ABB RobotStudio station: proiect_1301A_Nichifor_Cristian_Musteata_Valeriu.rspag

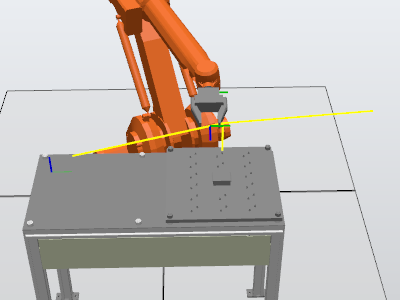
--- station ---
Station pikplace (saved by RobotStudio 25.4.11475.0)
Controller R1400, task T_ROB1: task frame (RAPID world) sits at (0, 0, 0) mm, rotated rx 0 ry 0 rz -45 deg in the station
Controller R1400
  mechanical unit ROB_1: IRB1400_5_144__01, 6 joints, base frame (0, 0, 0) mm
Layout (positions relative to the parent item):
  - IRB1400_5_144__01 [mechanism, from Robots\IRB1400_5_144__01.rslib] at (0, 0, 0) mm, rotated rx 0 ry 0 rz -45 deg; joint values [-0.3822, -0.6501, 0.0834, -1.4092, 0.4046, 1.4548] (rad or m)
  - Gripper_R1400 [smart component, from Components\Gripper_R1400.rslib] at (201.82, -557.27, 1000.36) mm, rotated rx 180 ry 81.97 rz 90 deg
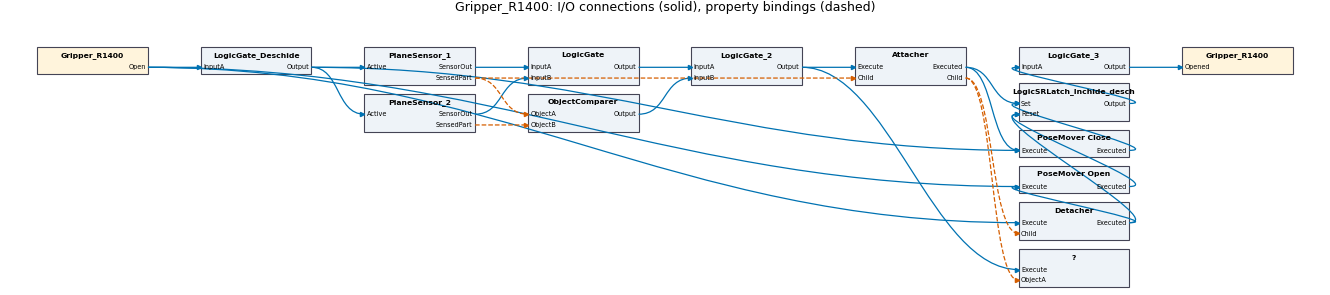
      connections:
        Attacher.Executed -> LogicSRLatch_Inchide_deschide.Set
        Detacher.Executed -> LogicSRLatch_Inchide_deschide.Reset
        Attacher.Executed -> PoseMover Close.Execute
        PoseMover Close.Executed -> LogicSRLatch_Inchide_deschide.Set
        Detacher.Executed -> PoseMover Open.Execute
        PoseMover Open.Executed -> LogicSRLatch_Inchide_deschide.Reset
        LogicGate.Output -> LogicGate_2.InputA
        ObjectComparer.Output -> LogicGate_2.InputB
        LogicGate_2.Output -> ?.Execute
        LogicGate_2.Output -> Attacher.Execute
        PlaneSensor_1.SensorOut -> LogicGate.InputA
        PlaneSensor_2.SensorOut -> LogicGate.InputB
        LogicGate_Deschide.Output -> PlaneSensor_2.Active
        LogicGate_Deschide.Output -> PlaneSensor_1.Active
        LogicGate_Deschide.Output -> PoseMover Close.Execute
        LogicSRLatch_Inchide_deschide.Output -> LogicGate_3.InputA
        LogicGate_3.Output -> Gripper_R1400.Opened
        Gripper_R1400.Open -> LogicGate_Deschide.InputA
        Gripper_R1400.Open -> Detacher.Execute
        Gripper_R1400.Open -> PoseMover Open.Execute
        Attacher.Child => Detacher.Child
        Attacher.Child => ?.ObjectA
        PlaneSensor_1.SensedPart => Attacher.Child
        PlaneSensor_1.SensedPart => ObjectComparer.ObjectA
        PlaneSensor_2.SensedPart => ObjectComparer.ObjectB
    - Attacher [smart component, from Components\Gripper_R1400.rslib]
        properties: Parent=Gripper; Flange=0; Child=(none); Mount=false; Offset=[0 0 0]; Orientation=[0 0 0]
    - Detacher [smart component, from Components\Gripper_R1400.rslib]
        properties: Child=(none); KeepPosition=true
    - LogicGate_Deschide [smart component, from Components\Gripper_R1400.rslib]
        properties: Operator=NOT; Delay=0
    - LogicSRLatch_Inchide_deschide [smart component, from Components\Gripper_R1400.rslib]
    - PoseMover Close [smart component, from Components\Gripper_R1400.rslib]
        properties: Mechanism=Gripper; Pose=3; Duration=0
    - PoseMover Open [smart component, from Components\Gripper_R1400.rslib]
        properties: Mechanism=Gripper; Pose=2; Duration=0
    - ObjectComparer [smart component, from Components\ObjectComparer.rslib]
        properties: ObjectA=(none); ObjectB=(none)
    - LogicGate [smart component, from Components\LogicGate.rslib]
        properties: Operator=AND; Delay=0
    - LogicGate_2 [smart component, from Components\LogicGate.rslib]
        properties: Operator=AND; Delay=0
    - PlaneSensor_1 [smart component, from Components\PlaneSensor.rslib]
        properties: Origin=[-0.015 0.03 0.128]; Axis1=[0 0 0.055]; Axis2=[0.03 0 0]; SensedPart=(none); SenseMultiple=false; Tag=(none)
      - _sensorPart_ [part], size 30 x 0 x 55 mm
    - PlaneSensor_2 [smart component, from Components\PlaneSensor.rslib]
        properties: Origin=[-0.015 -0.03 0.128]; Axis1=[0 0 0.055]; Axis2=[0.03 0 0]; SensedPart=(none); SenseMultiple=false; Tag=(none)
      - _sensorPart_ [part], size 30 x 0 x 55 mm
    - Gripper [mechanism, from Components\Gripper_R1400.rslib] at (0, 0.03, 0) mm; joint values [0.0105, -0.0105] (rad or m)
    - LogicGate_3 [smart component, from Components\LogicGate.rslib]
        properties: Operator=NOT; Delay=0
  - Paleta [part, from Components\Paleta.rslib] at (240, -878, 808) mm, rotated rx 0 ry 0 rz -90 deg
  - Stoc1400 [smart component, from Components\Stoc1400.rslib] at (0, -878, 0) mm, rotated rx 0 ry 0 rz -90 deg
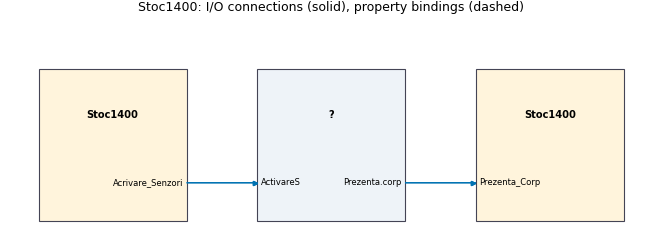
      connections:
        Stoc1400.Acrivare_Senzori -> ?.ActivareS
        Stoc1400.Acrivare_Senzori -> ?.ActivareS
        ?.Prezenta.corp -> Stoc1400.Prezenta_Corp
        ?.Prezenta.corp -> Stoc1400.Prezenta_Corp
    - 679#Body 1 [part, from Components\Stoc1400.rslib]
    - 681#Body 2 [part, from Components\Stoc1400.rslib]
    - 683#Body 3 [part, from Components\Stoc1400.rslib]
    - 685#Body 4 [part, from Components\Stoc1400.rslib]
    - 687#Body 5 [part, from Components\Stoc1400.rslib]
    - 689#Body 6 [part, from Components\Stoc1400.rslib]
    - 691#Body 7 [part, from Components\Stoc1400.rslib]
    - 693#Body 8 [part, from Components\Stoc1400.rslib]
    - 695#Body 9 [part, from Components\Stoc1400.rslib]
    - 697#Body 10 [part, from Components\Stoc1400.rslib]
    - 701#Body 12 [part, from Components\Stoc1400.rslib]
    - 703#Body 13 [part, from Components\Stoc1400.rslib]
    - 705#Body 14 [part, from Components\Stoc1400.rslib]
    - 707#Body 15 [part, from Components\Stoc1400.rslib]
    - 755#Body 39 [part, from Components\Stoc1400.rslib]
    - 757#Body 40 [part, from Components\Stoc1400.rslib]
    - 759#Body 41 [part, from Components\Stoc1400.rslib]
    - 761#Body 42 [part, from Components\Stoc1400.rslib]
    - 785#Body 54 [part, from Components\Stoc1400.rslib]
    - 787#Body 55 [part, from Components\Stoc1400.rslib]
    - 789#Body 56 [part, from Components\Stoc1400.rslib]
    - 791#Body 57 [part, from Components\Stoc1400.rslib]
    - 793#Body 58 [part, from Components\Stoc1400.rslib]
    - Part [part, from Components\Stoc1400.rslib]
    - Part_2 [part, from Components\Stoc1400.rslib]
    - Part_3 [part, from Components\Stoc1400.rslib]
    - Part_4 [part, from Components\Stoc1400.rslib]
Attachment: Gripper_R1400 is attached to IRB1400_5_144__01 / Link6
Station logic (signal -> signal, property => property):
  R1400.DO10_9 -> Gripper_R1400.Open
Targets, tools, work objects and paths stored in the station and not in the controller backup, written as RAPID:
! task T_ROB1
MODULE Module1
  PROC ZERO()
    MoveL T0_1,v200,fine,Efector\WObj:=Workobject_1;
    MoveC T0_2,T0_3,v200,fine,Efector\WObj:=Workobject_1;
    MoveC T0_4,T0_1,v200,fine,Efector\WObj:=Workobject_1;
    MoveL ref,v200,fine,Efector\WObj:=Workobject_1;
  ENDPROC
  PROC ONE()
    MoveL T1_1,v200,fine,Efector\WObj:=Workobject_1;
    MoveL T1_2,v200,fine,Efector\WObj:=Workobject_1;
    MoveL T1_3,v200,fine,Efector\WObj:=Workobject_1;
    MoveL ref,v200,fine,Efector\WObj:=Workobject_1;
  ENDPROC
  PROC TWO()
    MoveL T2_1,v200,fine,Efector\WObj:=Workobject_1;
    MoveC T2_2,T2_3,v200,fine,Efector\WObj:=Workobject_1;
    MoveL T2_4,v200,fine,Efector\WObj:=Workobject_1;
    MoveL T2_5,v200,fine,Efector\WObj:=Workobject_1;
    MoveL ref,v200,fine,Efector\WObj:=Workobject_1;
  ENDPROC
  PROC THREE()
    MoveL T3_1,v200,fine,Efector\WObj:=Workobject_1;
    MoveL T3_2,v200,fine,Efector\WObj:=Workobject_1;
    MoveL T3_3,v200,fine,Efector\WObj:=Workobject_1;
    MoveC T3_4,T3_5,v200,fine,Efector\WObj:=Workobject_1;
    MoveL ref,v200,fine,Efector\WObj:=Workobject_1;
  ENDPROC
  PROC FOUR()
    MoveL T4_1,v200,fine,Efector\WObj:=Workobject_1;
    MoveL T4_2,v200,fine,Efector\WObj:=Workobject_1;
    MoveL T4_3,v200,fine,Efector\WObj:=Workobject_1;
    MoveL T4_4,v200,fine,Efector\WObj:=Workobject_1;
    MoveL ref,v200,fine,Efector\WObj:=Workobject_1;
  ENDPROC
  PROC NINE()
    MoveL T9_1,v200,fine,Efector\WObj:=Workobject_1;
    MoveC T9_2,T9_3,v200,fine,Efector\WObj:=Workobject_1;
    MoveL T9_4,v200,fine,Efector\WObj:=Workobject_1;
    MoveC T9_5,T9_6,v200,fine,Efector\WObj:=Workobject_1;
    MoveC T9_7,T9_4,v200,fine,Efector\WObj:=Workobject_1;
    MoveL ref,v200,fine,Efector\WObj:=Workobject_1;
  ENDPROC
  PROC SIX()
    MoveL T6_1,v200,fine,Efector\WObj:=Workobject_1;
    MoveC T6_2,T6_3,v200,fine,Efector\WObj:=Workobject_1;
    MoveL T6_4,v200,fine,Efector\WObj:=Workobject_1;
    MoveC T6_5,T6_6,v200,fine,Efector\WObj:=Workobject_1;
    MoveC T6_7,T6_4,v200,fine,Efector\WObj:=Workobject_1;
    MoveL ref,v200,fine,Efector\WObj:=Workobject_1;
  ENDPROC
  PROC FIVE()
    MoveL T5_1,v200,fine,Efector\WObj:=Workobject_1;
    MoveL T5_2,v200,fine,Efector\WObj:=Workobject_1;
    MoveL T5_3,v200,fine,Efector\WObj:=Workobject_1;
    MoveC T5_4,T5_5,v200,fine,Efector\WObj:=Workobject_1;
    MoveL ref,v200,fine,Efector\WObj:=Workobject_1;
  ENDPROC
  PROC SEVEN()
    MoveL T7_1,v200,fine,Efector\WObj:=Workobject_1;
    MoveL T7_2,v200,fine,Efector\WObj:=Workobject_1;
    MoveL T7_3,v200,fine,Efector\WObj:=Workobject_1;
    MoveL ref,v200,fine,Efector\WObj:=Workobject_1;
  ENDPROC
  PROC EIGHT()
    MoveL T8_1,v200,fine,Efector\WObj:=Workobject_1;
    MoveC T8_2,T8_3,v200,fine,Efector\WObj:=Workobject_1;
    MoveC T8_4,T8_5,v200,fine,Efector\WObj:=Workobject_1;
    MoveC T8_6,T8_3,v200,fine,Efector\WObj:=Workobject_1;
    MoveC T8_7,T8_1,v200,fine,Efector\WObj:=Workobject_1;
    MoveL ref,v200,fine,Efector\WObj:=Workobject_1;
  ENDPROC
ENDMODULE


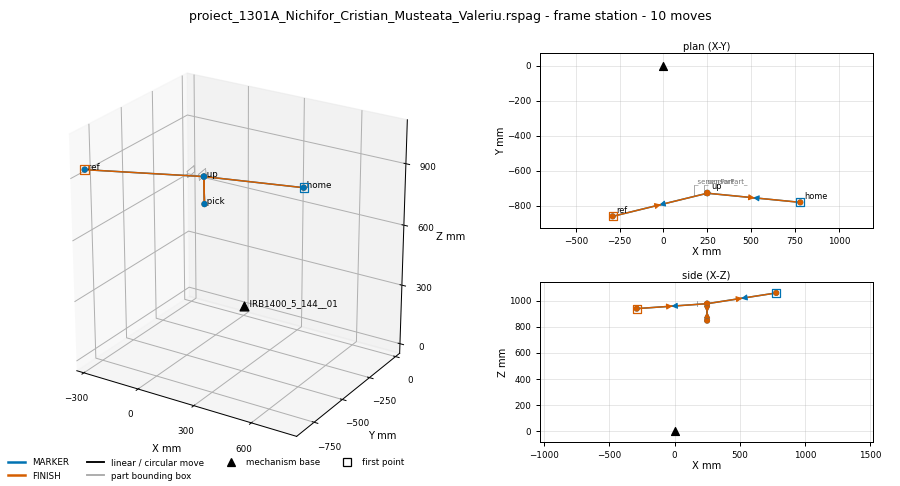
[picture p0: tool path of proiect_1301A_Nichifor_Cristian_Musteata_Valeriu.rspag in frame station, 10 of 60 moves have a stored position in this frame; points joined in program order, loops and branches not executed]
--- Controller Data/R1400/RAPID/TASK1/PROGMOD/Module1.mod ---
MODULE Module1
    PERS tooldata Efector:=[TRUE,[[0,0.033033672,184.3],[1,0,0,0]],[1.5,[0,0,90],[1,0,0,0],0.01,0.01,0.01]];
    PERS wobjdata Workobject_1:=[FALSE,TRUE,"",[[276.123735704,-827.667234537,798.663444233],[0.923877305,0.000104396,-0.002651392,-0.382679612]],[[0,0,0],[1,0,0,0]]];
    CONST robtarget home:=[[0.834488103,1170.696929347,259.084700159],[0.459642479,-0.331462463,0.801426912,0.191249396],[-1,0,-1,0],[9E+09,9E+09,9E+09,9E+09,9E+09,9E+09]];
    CONST robtarget up:=[[-51.633208179,640.397645531,178.164826806],[0.705400436,-0.000783768,0.708808148,-0.000787554],[-1,-2,1,0],[9E+09,9E+09,9E+09,9E+09,9E+09,9E+09]];
    CONST robtarget pick:=[[-55.259706896,640.108764023,48.166657408],[0.705400436,-0.000783768,0.708808148,-0.000787554],[-1,-2,1,0],[9E+09,9E+09,9E+09,9E+09,9E+09,9E+09]];
    CONST robtarget ref:=[[80.028130577,100.720123453,140.72904745],[0.002409616,-0.000002677,-0.99999648,0.001111092],[-1,0,-1,0],[9E+09,9E+09,9E+09,9E+09,9E+09,9E+09]];
CONST robtarget T0_1:=[[9.546208479,100.497907125,40.730455604],[0.002409616,-0.000002677,-0.99999648,0.001111092],[-1,-1,0,0],[9E+09,9E+09,9E+09,9E+09,9E+09,9E+09]];
    CONST robtarget T0_2:=[[41.035842809,79.777621062,40.624742502],[0.002409616,-0.000002677,-0.99999648,0.001111092],[-1,-1,0,0],[9E+09,9E+09,9E+09,9E+09,9E+09,9E+09]];
    CONST robtarget T0_3:=[[81.732370203,107.749116179,40.366456021],[0.002409616,-0.000002677,-0.99999648,0.001111092],[-1,-1,0,0],[9E+09,9E+09,9E+09,9E+09,9E+09,9E+09]];
    CONST robtarget T0_4:=[[36.187899089,125.180560875,40.547211878],[0.002409616,-0.000002677,-0.99999648,0.001111092],[-1,-1,0,0],[9E+09,9E+09,9E+09,9E+09,9E+09,9E+09]];
    CONST robtarget T1_1:=[[23.778043214,86.267789909,40.693490346],[0.002409616,-0.000002677,-0.99999648,0.001111093],[-1,0,-1,0],[9E+09,9E+09,9E+09,9E+09,9E+09,9E+09]];
    CONST robtarget T1_2:=[[8.731217939,99.845917516,40.735832074],[0.002409616,-0.000002677,-0.99999648,0.001111093],[-1,0,-1,0],[9E+09,9E+09,9E+09,9E+09,9E+09,9E+09]];
    CONST robtarget T1_3:=[[80.636382929,100.842145042,40.387086501],[0.002409616,-0.000002677,-0.99999648,0.001111093],[-1,0,-1,0],[9E+09,9E+09,9E+09,9E+09,9E+09,9E+09]];
    CONST robtarget T2_1:=[[31.755950553,80.841717855,40.667100297],[0.002409616,-0.000002677,-0.99999648,0.001111093],[-1,0,-1,0],[9E+09,9E+09,9E+09,9E+09,9E+09,9E+09]];
    CONST robtarget T2_2:=[[6.08624864,99.311947147,40.74976553],[0.002409616,-0.000002677,-0.99999648,0.001111093],[-1,0,-1,0],[9E+09,9E+09,9E+09,9E+09,9E+09,9E+09]];
    CONST robtarget T2_3:=[[29.104981321,125.470636052,40.580701845],[0.002409616,-0.000002677,-0.99999648,0.001111093],[-1,0,-1,0],[9E+09,9E+09,9E+09,9E+09,9E+09,9E+09]];
    CONST robtarget T2_4:=[[71.480489244,86.448278602,40.463197375],[0.002409616,-0.000002677,-0.99999648,0.001111093],[-1,0,-1,0],[9E+09,9E+09,9E+09,9E+09,9E+09,9E+09]];
    CONST robtarget T2_5:=[[70.80349709,127.872183573,40.374407927],[0.002409616,-0.000002677,-0.99999648,0.001111093],[-1,0,-1,0],[9E+09,9E+09,9E+09,9E+09,9E+09,9E+09]];
    CONST robtarget T3_1:=[[18.710215411,82.591773594,40.726082499],[0.002409616,-0.000002677,-0.99999648,0.001111093],[-1,0,-1,0],[9E+09,9E+09,9E+09,9E+09,9E+09,9E+09]];
    CONST robtarget T3_2:=[[19.688090682,111.187772163,40.657823899],[0.002409616,-0.000002677,-0.99999648,0.001111093],[-1,0,-1,0],[9E+09,9E+09,9E+09,9E+09,9E+09,9E+09]];
    CONST robtarget T3_3:=[[45.419791871,103.366515913,40.55119576],[0.002409616,-0.000002677,-0.99999648,0.001111093],[-1,0,-1,0],[9E+09,9E+09,9E+09,9E+09,9E+09,9E+09]];
    CONST robtarget T3_4:=[[68.022529389,116.554241299,40.41296091],[0.002409616,-0.000002677,-0.99999648,0.001111093],[-1,0,-1,0],[9E+09,9E+09,9E+09,9E+09,9E+09,9E+09]];
    CONST robtarget T3_5:=[[73.635464218,90.505245507,40.443796548],[0.002409616,-0.000002677,-0.99999648,0.001111093],[-1,0,-1,0],[9E+09,9E+09,9E+09,9E+09,9E+09,9E+09]];
    CONST robtarget T4_1:=[[53.83069419,124.165374487,40.464442032],[0.002409616,-0.000002677,-0.99999648,0.001111093],[-1,0,-1,0],[9E+09,9E+09,9E+09,9E+09,9E+09,9E+09]];
    CONST robtarget T4_2:=[[53.075702975,80.033491537,40.566150282],[0.002409616,-0.000002677,-0.99999648,0.001111093],[-1,0,-1,0],[9E+09,9E+09,9E+09,9E+09,9E+09,9E+09]];
    CONST robtarget T4_3:=[[9.18787321,109.525888713,40.712120516],[0.002409616,-0.000002677,-0.99999648,0.001111093],[-1,0,-1,0],[9E+09,9E+09,9E+09,9E+09,9E+09,9E+09]];
    CONST robtarget T4_4:=[[83.035355052,110.99609425,40.352961057],[0.002409616,-0.000002677,-0.99999648,0.001111093],[-1,0,-1,0],[9E+09,9E+09,9E+09,9E+09,9E+09,9E+09]];
    CONST robtarget T9_1:=[[70.611499337,82.764297004,40.475571821],[0.002409616,-0.000002677,-0.99999648,0.001111093],[-1,0,-1,0],[9E+09,9E+09,9E+09,9E+09,9E+09,9E+09]];
    CONST robtarget T9_2:=[[86.448315421,103.968075054,40.352130656],[0.002409616,-0.000002677,-0.99999648,0.001111093],[-1,0,-1,0],[9E+09,9E+09,9E+09,9E+09,9E+09,9E+09]];
    CONST robtarget T9_3:=[[68.016529456,122.326227112,40.400163337],[0.002409616,-0.000002677,-0.99999648,0.001111093],[-1,0,-1,0],[9E+09,9E+09,9E+09,9E+09,9E+09,9E+09]];
    CONST robtarget T9_4:=[[40.69684671,123.155517631,40.529981942],[0.002409616,-0.000002677,-0.99999648,0.001111093],[-1,0,-1,0],[9E+09,9E+09,9E+09,9E+09,9E+09,9E+09]];
    CONST robtarget T9_5:=[[20.029086726,101.021793612,40.678771345],[0.002409616,-0.000002677,-0.99999648,0.001111093],[-1,0,-1,0],[9E+09,9E+09,9E+09,9E+09,9E+09,9E+09]];
    CONST robtarget T9_6:=[[37.315885986,84.371649598,40.632461157],[0.002409616,-0.000002677,-0.99999648,0.001111093],[-1,0,-1,0],[9E+09,9E+09,9E+09,9E+09,9E+09,9E+09]];
    CONST robtarget T9_7:=[[49.971739012,101.45747188,40.533500882],[0.002409616,-0.000002677,-0.99999648,0.001111093],[-1,0,-1,0],[9E+09,9E+09,9E+09,9E+09,9E+09,9E+09]];
    CONST robtarget T6_1:=[[29.037119424,125.16526603,40.581707484],[0.002409616,0.000002677,-0.99999648,0.001111093],[-1,-1,-1,0],[9E+09,9E+09,9E+09,9E+09,9E+09,9E+09]];
    CONST robtarget T6_2:=[[13.20030334,103.96148798,40.705148627],[0.002409616,0.000002677,-0.99999648,0.001111093],[-1,-1,-1,0],[9E+09,9E+09,9E+09,9E+09,9E+09,9E+09]];
    CONST robtarget T6_3:=[[31.632089305,85.603335922,40.657115952],[0.002409616,0.000002677,-0.99999648,0.001111093],[-1,-1,-1,0],[9E+09,9E+09,9E+09,9E+09,9E+09,9E+09]];
    CONST robtarget T6_4:=[[58.951772051,84.774045403,40.527297366],[0.002409616,0.000002677,-0.99999648,0.001111093],[-1,-1,-1,0],[9E+09,9E+09,9E+09,9E+09,9E+09,9E+09]];
    CONST robtarget T6_5:=[[79.619532035,106.907769422,40.378507987],[0.002409616,0.000002677,-0.99999648,0.001111093],[-1,-1,-1,0],[9E+09,9E+09,9E+09,9E+09,9E+09,9E+09]];
    CONST robtarget T6_6:=[[62.332732775,123.557913436,40.424818171],[0.002409616,0.000002677,-0.99999648,0.001111093],[-1,-1,-1,0],[9E+09,9E+09,9E+09,9E+09,9E+09,9E+09]];
    CONST robtarget T6_7:=[[44.189479584,106.472149918,40.550223668],[0.002409616,0.000002677,-0.99999648,0.001111093],[-1,-1,-1,0],[9E+09,9E+09,9E+09,9E+09,9E+09,9E+09]];
    CONST robtarget T5_1:=[[17.47494015,121.068036328,40.646533482],[0.002409616,-0.000002677,-0.99999648,0.001111092],[-1,0,-1,0],[9E+09,9E+09,9E+09,9E+09,9E+09,9E+09]];
    CONST robtarget T5_2:=[[17.358941509,85.796124659,40.725473626],[0.002409616,-0.000002677,-0.99999648,0.001111092],[-1,0,-1,0],[9E+09,9E+09,9E+09,9E+09,9E+09,9E+09]];
    CONST robtarget T5_3:=[[38.084700828,86.30490145,40.62445961],[0.002409616,-0.000002677,-0.99999648,0.001111092],[-1,0,-1,0],[9E+09,9E+09,9E+09,9E+09,9E+09,9E+09]];
    CONST robtarget T5_4:=[[56.476487242,111.192166678,40.480519899],[0.002409616,-0.000002677,-0.99999648,0.001111092],[-1,0,-1,0],[9E+09,9E+09,9E+09,9E+09,9E+09,9E+09]];
    CONST robtarget T5_5:=[[73.027295052,86.419526967,40.455806449],[0.002409616,-0.000002677,-0.99999648,0.001111092],[-1,0,-1,0],[9E+09,9E+09,9E+09,9E+09,9E+09,9E+09]];
    CONST robtarget T7_1:=[[18.254137879,83.451889647,40.726368808],[0.002409616,-0.000002677,-0.99999648,0.001111092],[-1,0,-1,0],[9E+09,9E+09,9E+09,9E+09,9E+09,9E+09]];
    CONST robtarget T7_2:=[[16.933153208,115.512476931,40.661490103],[0.002409616,-0.000002677,-0.99999648,0.001111092],[-1,0,-1,0],[9E+09,9E+09,9E+09,9E+09,9E+09,9E+09]];
    CONST robtarget T7_3:=[[75.380474485,98.997889493,40.416514244],[0.002409616,-0.000002677,-0.99999648,0.001111092],[-1,0,-1,0],[9E+09,9E+09,9E+09,9E+09,9E+09,9E+09]];
    CONST robtarget T8_1:=[[78.856287686,108.091037322,40.379556329],[0.002409616,-0.000002677,-0.99999648,0.001111092],[-1,0,-1,0],[9E+09,9E+09,9E+09,9E+09,9E+09,9E+09]];
    CONST robtarget T8_2:=[[57.493535772,87.570316763,40.528110688],[0.002409616,-0.000002677,-0.99999648,0.001111092],[-1,0,-1,0],[9E+09,9E+09,9E+09,9E+09,9E+09,9E+09]];
    CONST robtarget T8_3:=[[41.951716246,106.624436154,40.560669208],[0.002409616,-0.000002677,-0.99999648,0.001111092],[-1,0,-1,0],[9E+09,9E+09,9E+09,9E+09,9E+09,9E+09]];
    CONST robtarget T8_4:=[[18.719986023,120.847649824,40.641022855],[0.002409616,-0.000002677,-0.99999648,0.001111092],[-1,0,-1,0],[9E+09,9E+09,9E+09,9E+09,9E+09,9E+09]];
    CONST robtarget T8_5:=[[-0.434791533,103.81389701,40.771187619],[0.002409616,-0.000002677,-0.99999648,0.001111092],[-1,0,-1,0],[9E+09,9E+09,9E+09,9E+09,9E+09,9E+09]];
    CONST robtarget T8_6:=[[20.170969186,87.149717488,40.708913585],[0.002409616,-0.000002677,-0.99999648,0.001111092],[-1,0,-1,0],[9E+09,9E+09,9E+09,9E+09,9E+09,9E+09]];
    CONST robtarget T8_7:=[[60.168504694,124.215197637,40.433787102],[0.002409616,-0.000002677,-0.99999648,0.001111092],[-1,0,-1,0],[9E+09,9E+09,9E+09,9E+09,9E+09,9E+09]];

    CONST num DIGIT_Y_STEP := 50;

    PROC main()
        MARKER;
        CalculatorC;
        FINISH;
    ENDPROC

    PROC CalculatorC()
        VAR num firstTerm;
        VAR num secondTerm;
        VAR num operation;
        VAR num result;

        TPErase;
        TPReadNum firstTerm, "Primul termen:";
        TPReadFK operation, "Alege operatia", "+", "-", "*", "/", "";
        TPReadNum secondTerm, "Al doilea termen:";

        IF operation = 1 THEN
            result := firstTerm + secondTerm;
        ELSEIF operation = 2 THEN
            result := firstTerm - secondTerm;
        ELSEIF operation = 3 THEN
            result := firstTerm * secondTerm;
        ELSEIF operation = 4 THEN
            IF secondTerm = 0 THEN
                TPWrite "Eroare: impartire la 0.";
                RETURN;
            ENDIF
            result := firstTerm / secondTerm;
        ELSE
            TPWrite "Operatie invalida.";
            RETURN;
        ENDIF

        result := Trunc(result);

        IF result < 0 THEN
            TPWrite "Rezultat negativ. Desenez valoarea absoluta.";
            result := -result;
        ENDIF

        DrawNumber result;
    ENDPROC

    PROC DrawNumber(num value)
        VAR num n;
        VAR num divisor;
        VAR num digit;
        VAR num yOffset;

        n := Trunc(value);

        IF n = 0 THEN
            ZERO 0;
            RETURN;
        ENDIF

        divisor := 1;
        WHILE n >= divisor * 10 DO
            divisor := divisor * 10;
        ENDWHILE

        yOffset := 0;
        WHILE divisor >= 1 DO
            digit := Trunc(n / divisor);
            DrawDigit digit, yOffset;
            n := n - digit * divisor;
            divisor := divisor / 10;
            yOffset := yOffset + DIGIT_Y_STEP;
        ENDWHILE
    ENDPROC

    PROC DrawDigit(num digit, num yOffset)
        IF digit = 0 THEN
            ZERO yOffset;
        ELSEIF digit = 1 THEN
            ONE yOffset;
        ELSEIF digit = 2 THEN
            TWO yOffset;
        ELSEIF digit = 3 THEN
            THREE yOffset;
        ELSEIF digit = 4 THEN
            FOUR yOffset;
        ELSEIF digit = 5 THEN
            FIVE yOffset;
        ELSEIF digit = 6 THEN
            SIX yOffset;
        ELSEIF digit = 7 THEN
            SEVEN yOffset;
        ELSEIF digit = 8 THEN
            EIGHT yOffset;
        ELSEIF digit = 9 THEN
            NINE yOffset;
        ENDIF
    ENDPROC

    PROC ZERO(num yOffset)
        MoveL Offs(T0_1,0,yOffset,0),v200,fine,Efector\WObj:=Workobject_1;
        MoveC Offs(T0_2,0,yOffset,0),Offs(T0_3,0,yOffset,0),v200,fine,Efector\WObj:=Workobject_1;
        MoveC Offs(T0_4,0,yOffset,0),Offs(T0_1,0,yOffset,0),v200,fine,Efector\WObj:=Workobject_1;
        MoveL Offs(ref,0,yOffset,0),v200,fine,Efector\WObj:=Workobject_1;
    ENDPROC
    PROC MARKER()
        Set DO10_9;
        MoveL home,v200,fine,Efector\WObj:=Workobject_1;
        MoveL up,v200,fine,Efector\WObj:=Workobject_1;
        MoveL pick,v200,fine,Efector\WObj:=Workobject_1;
        Reset DO10_9;
        WaitTime 2;
        MoveL up,v200,fine,Efector\WObj:=Workobject_1;
        WaitTime 2;
        MoveL ref,v200,fine,Efector\WObj:=Workobject_1;
    ENDPROC
    PROC FINISH()
        MoveL ref,v200,fine,Efector\WObj:=Workobject_1;
        MoveL up,v200,fine,Efector\WObj:=Workobject_1;
        MoveL pick,v200,fine,Efector\WObj:=Workobject_1;
        WaitTime 2;
        Set DO10_9;
        WaitTime 2;
        MoveL up,v200,fine,Efector\WObj:=Workobject_1;
        MoveL home,v200,fine,Efector\WObj:=Workobject_1;
    ENDPROC
    PROC ONE(num yOffset)
        MoveL Offs(T1_1,0,yOffset,0),v200,fine,Efector\WObj:=Workobject_1;
        MoveL Offs(T1_2,0,yOffset,0),v200,fine,Efector\WObj:=Workobject_1;
        MoveL Offs(T1_3,0,yOffset,0),v200,fine,Efector\WObj:=Workobject_1;
        MoveL Offs(ref,0,yOffset,0),v200,fine,Efector\WObj:=Workobject_1;
    ENDPROC
    PROC TWO(num yOffset)
        MoveL Offs(T2_1,0,yOffset,0),v200,fine,Efector\WObj:=Workobject_1;
        MoveC Offs(T2_2,0,yOffset,0),Offs(T2_3,0,yOffset,0),v200,fine,Efector\WObj:=Workobject_1;
        MoveL Offs(T2_4,0,yOffset,0),v200,fine,Efector\WObj:=Workobject_1;
        MoveL Offs(T2_5,0,yOffset,0),v200,fine,Efector\WObj:=Workobject_1;
        MoveL Offs(ref,0,yOffset,0),v200,fine,Efector\WObj:=Workobject_1;
    ENDPROC
    PROC THREE(num yOffset)
        MoveL Offs(T3_1,0,yOffset,0),v200,fine,Efector\WObj:=Workobject_1;
        MoveL Offs(T3_2,0,yOffset,0),v200,fine,Efector\WObj:=Workobject_1;
        MoveL Offs(T3_3,0,yOffset,0),v200,fine,Efector\WObj:=Workobject_1;
        MoveC Offs(T3_4,0,yOffset,0),Offs(T3_5,0,yOffset,0),v200,fine,Efector\WObj:=Workobject_1;
        MoveL Offs(ref,0,yOffset,0),v200,fine,Efector\WObj:=Workobject_1;
    ENDPROC
    PROC FOUR(num yOffset)
        MoveL Offs(T4_1,0,yOffset,0),v200,fine,Efector\WObj:=Workobject_1;
        MoveL Offs(T4_2,0,yOffset,0),v200,fine,Efector\WObj:=Workobject_1;
        MoveL Offs(T4_3,0,yOffset,0),v200,fine,Efector\WObj:=Workobject_1;
        MoveL Offs(T4_4,0,yOffset,0),v200,fine,Efector\WObj:=Workobject_1;
        MoveL Offs(ref,0,yOffset,0),v200,fine,Efector\WObj:=Workobject_1;
    ENDPROC
    PROC NINE(num yOffset)
        MoveL Offs(T9_1,0,yOffset,0),v200,fine,Efector\WObj:=Workobject_1;
        MoveC Offs(T9_2,0,yOffset,0),Offs(T9_3,0,yOffset,0),v200,fine,Efector\WObj:=Workobject_1;
        MoveL Offs(T9_4,0,yOffset,0),v200,fine,Efector\WObj:=Workobject_1;
        MoveC Offs(T9_5,0,yOffset,0),Offs(T9_6,0,yOffset,0),v200,fine,Efector\WObj:=Workobject_1;
        MoveC Offs(T9_7,0,yOffset,0),Offs(T9_4,0,yOffset,0),v200,fine,Efector\WObj:=Workobject_1;
        MoveL Offs(ref,0,yOffset,0),v200,fine,Efector\WObj:=Workobject_1;
    ENDPROC
    PROC SIX(num yOffset)
        MoveL Offs(T6_1,0,yOffset,0),v200,fine,Efector\WObj:=Workobject_1;
        MoveC Offs(T6_2,0,yOffset,0),Offs(T6_3,0,yOffset,0),v200,fine,Efector\WObj:=Workobject_1;
        MoveL Offs(T6_4,0,yOffset,0),v200,fine,Efector\WObj:=Workobject_1;
        MoveC Offs(T6_5,0,yOffset,0),Offs(T6_6,0,yOffset,0),v200,fine,Efector\WObj:=Workobject_1;
        MoveC Offs(T6_7,0,yOffset,0),Offs(T6_4,0,yOffset,0),v200,fine,Efector\WObj:=Workobject_1;
        MoveL Offs(ref,0,yOffset,0),v200,fine,Efector\WObj:=Workobject_1;
    ENDPROC
    PROC FIVE(num yOffset)
        MoveL Offs(T5_1,0,yOffset,0),v200,fine,Efector\WObj:=Workobject_1;
        MoveL Offs(T5_2,0,yOffset,0),v200,fine,Efector\WObj:=Workobject_1;
        MoveL Offs(T5_3,0,yOffset,0),v200,fine,Efector\WObj:=Workobject_1;
        MoveC Offs(T5_4,0,yOffset,0),Offs(T5_5,0,yOffset,0),v200,fine,Efector\WObj:=Workobject_1;
        MoveL Offs(ref,0,yOffset,0),v200,fine,Efector\WObj:=Workobject_1;
    ENDPROC
    PROC SEVEN(num yOffset)
        MoveL Offs(T7_1,0,yOffset,0),v200,fine,Efector\WObj:=Workobject_1;
        MoveL Offs(T7_2,0,yOffset,0),v200,fine,Efector\WObj:=Workobject_1;
        MoveL Offs(T7_3,0,yOffset,0),v200,fine,Efector\WObj:=Workobject_1;
        MoveL Offs(ref,0,yOffset,0),v200,fine,Efector\WObj:=Workobject_1;
    ENDPROC
    PROC EIGHT(num yOffset)
        MoveL Offs(T8_1,0,yOffset,0),v200,fine,Efector\WObj:=Workobject_1;
        MoveC Offs(T8_2,0,yOffset,0),Offs(T8_3,0,yOffset,0),v200,fine,Efector\WObj:=Workobject_1;
        MoveC Offs(T8_4,0,yOffset,0),Offs(T8_5,0,yOffset,0),v200,fine,Efector\WObj:=Workobject_1;
        MoveC Offs(T8_6,0,yOffset,0),Offs(T8_3,0,yOffset,0),v200,fine,Efector\WObj:=Workobject_1;
        MoveC Offs(T8_7,0,yOffset,0),Offs(T8_1,0,yOffset,0),v200,fine,Efector\WObj:=Workobject_1;
        MoveL Offs(ref,0,yOffset,0),v200,fine,Efector\WObj:=Workobject_1;
    ENDPROC

ENDMODULE

--- Controller Data/R1400/SYSPAR/EIO.cfg ---
EIO:CFG_1.0:5:60::
#
EIO_BUS:

      -Name "Virtual1"
#
EIO_UNIT_TYPE:

      -Name "Virtual" -VendorName "ABB" -ProductName "Virtual unit"
#
EIO_UNIT:

      -Name "TuIasi" -UnitType "Virtual" -Bus "Virtual1"
#
EIO_SIGNAL:

      -Name "DO10_9" -SignalType "DO" -Unit "TuIasi" -UnitMap "1" -Access "All"

      -Name "DO11_7" -SignalType "DO" -Unit "TuIasi" -UnitMap "2" -Access "All"

      -Name "DO11_8" -SignalType "DO" -Unit "TuIasi" -UnitMap "3" -Access "All"

      -Name "DO11_9" -SignalType "DO" -Unit "TuIasi" -UnitMap "4" -Access "All"

      -Name "DO12_1" -SignalType "DO" -Unit "TuIasi" -UnitMap "5" -Access "All"

      -Name "DO13_1" -SignalType "DO" -Unit "TuIasi" -UnitMap "7" -Access "All"

      -Name "DI11_9" -SignalType "DI" -Unit "TuIasi" -UnitMap "8" -Access "All"

      -Name "DI13_9" -SignalType "DI" -Unit "TuIasi" -UnitMap "9" -Access "All"

      -Name "AO12_1" -SignalType "AO" -Unit "TuIasi" -UnitMap "16-31"\
      -Access "All"

      -Name "DI12_2" -SignalType "DI" -Unit "TuIasi" -UnitMap "10" -Access "All"

      -Name "DO12_10" -SignalType "DO" -Unit "TuIasi" -UnitMap "11"\
      -Access "All"

      -Name "DI10_1" -SignalType "DI" -Unit "TuIasi" -UnitMap "12" -Access "All"

      -Name "DI10_7" -SignalType "DI" -Unit "TuIasi" -UnitMap "13" -Access "All"

      -Name "DI10_6" -SignalType "DI" -Unit "TuIasi" -UnitMap "14" -Access "All"

      -Name "DI10_5" -SignalType "DI" -Unit "TuIasi" -UnitMap "15" -Access "All"

      -Name "DI10_4" -SignalType "DI" -Unit "TuIasi" -UnitMap "32" -Access "All"

      -Name "DO10_3" -SignalType "DO" -Unit "TuIasi" -UnitMap "33" -Access "All"

      -Name "DO10_4" -SignalType "DO" -Unit "TuIasi" -UnitMap "34" -Access "All"

      -Name "DO10_2" -SignalType "DO" -Unit "TuIasi" -UnitMap "35" -Access "All"

      -Name "DO10_1" -SignalType "DO" -Unit "TuIasi" -UnitMap "36" -Access "All"
#
EIO_ACCESS:

      -Name "All" -Rapid  -LocalManual  -LocalAuto  -RemoteManual  -RemoteAuto
